{attribute addProperty BoxType "EP9128-0020-0016"}
{attribute addProperty Id "A_0004_EP9128_0021_0016A_0004_EP9128_0021_0016_B7B89D3D4614576.75A_0001_EP9128_0020_0016_2_EP9128_1020EP9128_179A0949162A_0001_EP9128_0020_0016_3_EP9128_2020EP9128_179A0949162"}
{attribute addProperty CRC "2144582397"}
{attribute addProperty SizeInBites "4646"}
{attribute addProperty SizeInBytes "580.75"}
TYPE A_0001_EP9128_0020_0016_7FD3BAFD EXTENDS EP9128_179A0949 :
STRUCT
	{attribute addProperty Name "A_0004_EP9128_0021_0016"}
	A_0004_EP9128_0021_0016 : A_0004_EP9128_0021_0016_B7B89D3D;
	{attribute addProperty Name "A_0001_EP9128_0020_0016_2_EP9128_1020"}
	A_0001_EP9128_0020_0016_2_EP9128_1020 : EP9128_179A0949;
	{attribute addProperty Name "A_0001_EP9128_0020_0016_3_EP9128_2020"}
	A_0001_EP9128_0020_0016_3_EP9128_2020 : EP9128_179A0949;
END_STRUCT
END_TYPE

(* stored: Version 1.2.0.0, ProductVersion 3.1.4024.9
   DUT A_0001_EP9128_0020_0016_7FD3BAFD: Id {15eecdc9-ebae-46e2-8cbf-674d266dc0a3} *)
